{attribute 'linkalways'} 
{attribute 'no_explicit_call' := 'This FB is a CLASS and must be accessed using methods or properties'}
{attribute 'enable_dynamic_creation'}
FUNCTION_BLOCK _ETcVnBlobCombination EXTENDS EnumDatatypeBase
VAR
	localData : ETcVnBlobCombination;
	activeData : REFERENCE TO ETcVnBlobCombination;
	enumBaseDatatype : _DINT(localData);
END_VAR

METHOD PRIVATE AddLocalEnumeration
VAR_INPUT
	Enumeration : T_MAXSTRING;
	Value : ETcVnBlobCombination;
END_VAR
AddEnumeration(Enumeration, Value);
END_METHOD

PROPERTY PUBLIC Address : PVOID
GET
Address := ADR(activeData);
END_GET
END_PROPERTY

METHOD PUBLIC ClearReference
VAR_INPUT
END_VAR
activeData REF= localData;
SetBaseDatatypeReference();
END_METHOD

METHOD PUBLIC Clone : I_Datatype
VAR
    pClone : POINTER TO _ETcVnBlobCombination;
END_VAR
pClone := __NEW(_ETcVnBlobCombination(InitialValue := Value));
Clone := pClone^;
END_METHOD

METHOD FB_init : BOOL
VAR_INPUT
	bInitRetains : BOOL; // if TRUE, the retain variables are initialized (warm start / cold start)
	bInCopyCode : BOOL;  // if TRUE, the instance afterwards gets moved into the copy code (online change)
	InitialValue : ETcVnBlobCombination;
END_VAR
localData := InitialValue;
AddBaseDatatype(enumBaseDatatype);
ClearReference();

AddLocalEnumeration('TCVN_BC_SMALLEST', ETcVnBlobCombination.TCVN_BC_SMALLEST);
AddLocalEnumeration('TCVN_BC_LARGEST', ETcVnBlobCombination.TCVN_BC_LARGEST);
AddLocalEnumeration('TCVN_BC_MIN_THRESHOLD', ETcVnBlobCombination.TCVN_BC_MIN_THRESHOLD);
AddLocalEnumeration('TCVN_BC_MAX_THRESHOLD', ETcVnBlobCombination.TCVN_BC_MAX_THRESHOLD);
AddLocalEnumeration('TCVN_BC_MEDIAN_THRESHOLD', ETcVnBlobCombination.TCVN_BC_MEDIAN_THRESHOLD);
END_METHOD

PROPERTY PUBLIC Identifier : T_MAXSTRING
GET
Identifier := 'ETcVnBlobCombination';
END_GET
END_PROPERTY

METHOD IsEnumeratorValueEqual : BOOL
VAR_INPUT
	Enumerator : I_KeyValueForwardEnumerator;
END_VAR
VAR
	storedValue : ETcVnBlobCombination;
END_VAR
IF NOT Enumerator.TryGet(storedValue) THEN
	RETURN;
END_IF

IsEnumeratorValueEqual := storedValue = activeData;
END_METHOD

METHOD PUBLIC MakeReferenceTo
VAR_INPUT
	ReferenceTarget : REFERENCE TO ETcVnBlobCombination;
END_VAR
activeData REF= ReferenceTarget;
SetBaseDatatypeReference();
END_METHOD

METHOD PROTECTED SetBaseDatatypeReference
VAR_INPUT
END_VAR
enumBaseDatatype.MakeReferenceTo(activeData);
END_METHOD

PROPERTY PUBLIC Size : UDINT
GET
Size := SIZEOF(activeData);
END_GET
END_PROPERTY

METHOD TryMakeReferenceTo : BOOL
VAR_INPUT
	Target : I_Datatype;
END_VAR
VAR
	targetAsEnum : I_EnumDatatype;
	pTargetData : POINTER TO ETcVnBlobCombination;
END_VAR
IF NOT Target.TryResolveAsEnumDatatype(targetAsEnum) THEN
	RETURN;
END_IF

IF targetAsEnum.Identifier <> Identifier THEN
	RETURN;
END_IF

pTargetData := Target.Address;
activeData REF= pTargetData^;
SetBaseDatatypeReference();
TryMakeReferenceTo := TRUE;
END_METHOD

PROPERTY PUBLIC Value : ETcVnBlobCombination
GET
Value := activeData;
END_GET
SET
activeData := Value;
END_SET
END_PROPERTY

END_FUNCTION_BLOCK

(* stored: Version 1.1.0.1, ProductVersion 3.1.4024.12
   POU _ETcVnBlobCombination: Id {503a463e-4570-4cf1-9f59-8f3556b39bb3}, SpecialFunc None
   Folder Constructor: Id {82898b2a-2300-4023-a403-00e6177523a1}
   Folder Private: Id {7e85741f-da45-44cb-b4d1-d51c645329fc}
   Folder Protected: Id {d0a758c8-3f5a-4a8d-a038-b9ef1ad87b48}
   Method AddLocalEnumeration: Id {497ddda5-ac97-4b54-a509-7d4e1973763a}
   Property Address: Id {82e8128f-1439-47e3-9c4a-86a228dc11c9}
   Get Get: Id {512f6045-c6c6-4728-a3e0-5d2afd1779ad}
   Method ClearReference: Id {cb2d5631-ff80-46d0-8a3a-29c9e814e46d}
   Method Clone: Id {aec6498b-3dab-471f-898b-770f277bed3d}
   Method FB_init: Id {1974410c-3a04-4b65-a5b3-4eb7b675d36e}
   Property Identifier: Id {5a8f1610-0def-480d-8d3a-fdbf0626b185}
   Get Get: Id {8b017a14-265c-4009-9524-ce2d09a33dff}
   Method IsEnumeratorValueEqual: Id {18fc3034-e12c-4041-84a6-e6684be85220}
   Method MakeReferenceTo: Id {dbbf2a36-f95b-4b13-9c10-0e07eaca15f6}
   Method SetBaseDatatypeReference: Id {00c013aa-58fd-4be1-b0df-462bbddf4724}
   Property Size: Id {ee9619a8-eccc-4f49-873c-549c412a0222}
   Get Get: Id {dc84db01-a622-48e0-898c-1a058882cd93}
   Method TryMakeReferenceTo: Id {9c328ecc-e122-497c-bbf5-eef3ad034208}
   Property Value: Id {53306e09-1240-40b8-a3ea-91d96898b00f}
   Get Get: Id {fb3b1242-2a69-4bd9-b17d-2107d5f1505b}
   Set Set: Id {d6d3ba50-d116-4298-b2e7-6a3a104dec1d} *)
